Staubli VAL3: moveStampUp.pgx

program moveStampUp(pointRs where, mdesc iniSpeed, trsf xyTrsf)
begin
  movej(appro(where, trUpThree*xyTrsf), tTool, iniSpeed)
  if iniSpeed == mExtremelySlow
    waitEndMove()
  endIf

  if iniSpeed == mExtremelySlow
    movej(appro(where, trZclose*xyTrsf), tTool, mVerySlow)
    waitEndMove()
  else
    movej(appro(where, trZclose*xyTrsf), tTool, mVerySlow)
  endIf

  movej(appro(where, trZsafe*xyTrsf), tTool, mSlow)
end
